// TIA Portal V17 export
// export: Created 2022-05-04T07:14:31.773887Z, ExportSetting WithDefaults, DisplayName Totally Integrated Automation Portal, DisplayVersion V17 Update 3, DisplayName TIA Portal Openness, DisplayVersion V17 Update 3, DisplayName TIA Portal Teamcenter Gateway, DisplayVersion V17 Update 3, DisplayName TIA Portal Version Control Interface, DisplayVersion V17, DisplayName SINAMICS Startdrive Advanced, DisplayVersion V17 Update2, DisplayName SINAMICS Startdrive G130, G150, S120, S150, SINAMICS MV, S210, DisplayVersion V17 Update2, DisplayName SINAMICS Startdrive G110M, G120, G120C, G120D, G120P, G115D, DisplayVersion V17 Update2, DisplayName STEP 7 Professional, DisplayVersion V17 Update 3, DisplayName STEP 7 CFC, DisplayVersion V17 Update 1, DisplayName STEP 7 Safety, DisplayVersion V17, DisplayName WinCC UA Professional, DisplayVersion V17 Update 3, DisplayName WinCC Unified Calendar, DisplayVersion V17, DisplayName WinCC Unified Performance Insight, DisplayVersion V17
TYPE "Connect_MODBUS_TCP"
// stored: IsFailsafeCompliant false
   STRUCT
      Connect : TCON_IP_v4;
   END_STRUCT;
   // Connect.InterfaceId := 64;
   // Connect.ID := 16#999;
   // Connect.ConnectionType := 11;
   // Connect.LocalPort := 502;
END_TYPE
